// TIA Portal V19 export
TYPE "LEXCHANGETRAY_typeHandlingXyzIoSignalControlNode"
// reset: Bool
// monitoring: LEXCHANGETRAY_typeHandlingXyzIoSignalContronNodeMonitoring
// stored: Access Published
   STRUCT
      reset : Bool;
      monitoring { S7_SetPoint := 'True'} : "LEXCHANGETRAY_typeHandlingXyzIoSignalContronNodeMonitoring";
   END_STRUCT;
END_TYPE
